TYPE ST_TestSystemDefaultParameters:
STRUCT
	aSetPointLimits	: ARRAY[1..2] OF REAL := [0,100];
END_STRUCT
END_TYPE

(* stored: Version 1.1.0.1, ProductVersion 3.1.4024.9
   DUT ST_TestSystemDefaultParameters: Id {4e04c00d-d74d-411b-98fb-73ed827f143f} *)
